// TIA Portal V19 export
VAR_GLOBAL   // PLC tag table "U2Em1"
END_VAR
VAR_GLOBAL CONSTANT   // user constants
   U2EM1_NO_OF_AXES : USInt := 1;   // Starts with 1. E.g., the value 4 means that 4 axes exist.
   U2EM1_JOB_EXECUTE : DInt := 100;   // ID for Job
   U2EM1_JOB_STOPPING : DInt := 200;
   U2EM1_JOB_HOLODING : DInt := 300;
   U2EM1_JOB_UNHOLODING : DInt := 400;
   U2EM1_JOB_RESTING : DInt := 500;
   U2EM1_JOB_STARTING : DInt := 600;
END_VAR
